// TIA Portal project "Stack_v000_000_005" (V16)
// 000_000_001: create project
// 000_000_002: create Stack.Add
// 000_000_003: create Stack.Remove
// 000_000_004: create Stack.Clear
// 000_000_005: create Stack
// 000_000_006: validation
// 001_000_000: release

(* hardware
DEVICE "S7-1200 station_1"  S7-1200 Station
   slot 0: "Rack_0"  S7-1200 Rack  Rack  V1.0
   slot 1: "PLC_1"  CPU 1212C DC/DC/DC  6ES7 212-1AE40-0XB0  V4.4
*)

// ===== PLC "PLC_1"  CPU 1212C DC/DC/DC =====

VAR_GLOBAL   // PLC tag table "Default tag table"
   "System_Byte" AT %MB1 : Byte;
   "FirstScan" AT %M1.0 : Bool;
   "DiagStatusUpdate" AT %M1.1 : Bool;
   "AlwaysTRUE" AT %M1.2 : Bool;
   "AlwaysFALSE" AT %M1.3 : Bool;
   "Clock_Byte" AT %MB0 : Byte;
   "Clock_10Hz" AT %M0.0 : Bool;
   "Clock_5Hz" AT %M0.1 : Bool;
   "Clock_2.5Hz" AT %M0.2 : Bool;
   "Clock_2Hz" AT %M0.3 : Bool;
   "Clock_1.25Hz" AT %M0.4 : Bool;
   "Clock_1Hz" AT %M0.5 : Bool;
   "Clock_0.625Hz" AT %M0.6 : Bool;
   "Clock_0.5Hz" AT %M0.7 : Bool;
END_VAR

TYPE "Int[+].UDT"
   STRUCT
      add : DInt;
      data : Array[0..4] of Int;
      length : DInt;
      remove : DInt := -1;
   END_STRUCT;
END_TYPE

TYPE "Stack.Calls.UDT"
   STRUCT
      idle : DInt;
      add : DInt := 1;
      remove : DInt := 2;
      clear : DInt := 3;
   END_STRUCT;
END_TYPE

ORGANIZATION_BLOCK "Main"   // OB1, LAD, ProgramCycle
TITLE = "Main Program Sweep (Cycle)"
{ S7_Optimized_Access := 'TRUE' }
VERSION : 0.1
   VAR_INPUT
      Initial_Call : Bool;   // Initial call of this OB
      Remanence : Bool;   // =True, if remanent data are available
   END_VAR
BEGIN
END_ORGANIZATION_BLOCK

// folder: Stack

FUNCTION_BLOCK "Stack"   // FB1, SCL
TITLE = Stack
{ S7_Optimized_Access := 'TRUE' }
AUTHOR : Machado
FAMILY : Stack
VERSION : 0.1
// calls:
//   idle = 0
//   add = 1
//   remove = 2
//   clear = 3
   VAR_INPUT
      call : DInt;
   END_VAR
   VAR_OUTPUT
      status : String;
   END_VAR
   VAR_IN_OUT
      value : Int;
   END_VAR
   VAR
      buffer : "Int[+].UDT";
      calls : "Stack.Calls.UDT";
   END_VAR
   VAR_TEMP
      message : String;
   END_VAR
   VAR CONSTANT
      IDLE_STATUS_MESSAGE : String := 'idle. no operation.';
      IDLE : DInt;
      ADD : DInt := 1;
      REMOVE : DInt := 2;
      CLEAR : DInt := 3;
      NULL_TOKEN : Int := -100;
      DEFAULT_ADD_INDEX : DInt := 0;
      DEFUALT_REMOVE_INDEX : DInt := -1;
   END_VAR
BEGIN
   CASE #call OF
       #IDLE:
           #message := #IDLE_STATUS_MESSAGE;
       #ADD:
           #message := "Stack.Add"(value := #value,
                                   buffer := #buffer);
       #REMOVE:
           #message := "Stack.Remove"(null_token := #NULL_TOKEN,
                                      value => #value,
                                      buffer := #buffer);
       #CLEAR:
           #message := "Stack.Clear"(default_add_index := #DEFAULT_ADD_INDEX,
                                     default_remove_index := #DEFUALT_REMOVE_INDEX,
                                     null_token := #NULL_TOKEN, buffer := #buffer);
       ELSE
           #message := #IDLE_STATUS_MESSAGE;
   END_CASE;
   #status := #message;
   RETURN;
END_FUNCTION_BLOCK

FUNCTION "Stack.Add" : String   // FC6, SCL
TITLE = Add a Value to the Stack
{ S7_Optimized_Access := 'TRUE' }
AUTHOR : Machado
FAMILY : Stack
VERSION : 0.1
// use [+].Push
// don't use [+].Add
   VAR_INPUT
      value : Int;
   END_VAR
   VAR_IN_OUT
      buffer : "Int[+].UDT";
   END_VAR
BEGIN
   #"Stack.Add" := "Int[+].Push"(value := #value,
                                 buffer := #buffer);
   RETURN;
END_FUNCTION

FUNCTION "Stack.Remove" : String   // FC8, SCL
TITLE = Remove a Value from a Stack
{ S7_Optimized_Access := 'TRUE' }
AUTHOR : Machado
FAMILY : Stack
VERSION : 0.1
// returns value and status message.
// use [+].Pop
// don't us [+].Remove
   VAR_INPUT
      null_token : Int;
   END_VAR
   VAR_OUTPUT
      value : Int;
   END_VAR
   VAR_IN_OUT
      buffer : "Int[+].UDT";
   END_VAR
BEGIN
   #"Stack.Remove" := "Int[+].Pop"(null_token := #null_token,
                                   value => #value,
                                   buffer := #buffer);
   RETURN;
END_FUNCTION

FUNCTION "Stack.Clear" : String   // FC10, SCL
TITLE = Clear All Values from a Stack
{ S7_Optimized_Access := 'TRUE' }
AUTHOR : Machado
FAMILY : Stack
VERSION : 0.1
// returns a string
   VAR_INPUT
      default_add_index : DInt;
      default_remove_index : DInt;
      null_token : Int;
   END_VAR
   VAR_IN_OUT
      buffer : "Int[+].UDT";
   END_VAR
BEGIN
   #"Stack.Clear" := "Int[+].Clear"(default_add_index := #default_add_index,
                                    default_remove_index := #default_remove_index,
                                    null_token := #null_token,
                                    buffer := #buffer);
   RETURN;
END_FUNCTION

// folder: Stack/Int[+]

FUNCTION "Int[+].IsFull" : Bool   // FC1, SCL
TITLE = Array Is Full
{ S7_Optimized_Access := 'TRUE' }
AUTHOR : Machado
FAMILY : Int[+]
VERSION : 0.1
// returns true if array is full
   VAR_INPUT
      buffer : "Int[+].UDT";
   END_VAR
   VAR_TEMP
      size : DInt;
   END_VAR
BEGIN
   #size := UDINT_TO_DINT("Int[].CountOfElements"(#buffer.data));
   IF #buffer.length = #size THEN
       #"Int[+].IsFull" := TRUE;
       RETURN;
   END_IF;
   #"Int[+].IsFull" := FALSE;
   RETURN;
END_FUNCTION

FUNCTION "Int[+].IsEmpty" : Bool   // FC3, SCL
TITLE = Int[+] Data Array Is Empty
{ S7_Optimized_Access := 'TRUE' }
AUTHOR : Machado
FAMILY : Int[+]
VERSION : 0.1
// returns true if array is empty
   VAR_INPUT
      buffer : "Int[+].UDT";
   END_VAR
BEGIN
   IF #buffer.length = 0 THEN
       #"Int[+].IsEmpty" := TRUE;
       RETURN;
   END_IF;
   #"Int[+].IsEmpty" := FALSE;
   RETURN;
END_FUNCTION

FUNCTION "Int[+].Push" : String   // FC4, SCL
TITLE = Push Value Into Data Array
{ S7_Optimized_Access := 'TRUE' }
AUTHOR : Machado
FAMILY : Int[+]
VERSION : 0.1
// dont use push with remove
   VAR_INPUT
      value : Int;
   END_VAR
   VAR_IN_OUT
      buffer : "Int[+].UDT";
   END_VAR
   VAR CONSTANT
      ARRAY_FULL : String := 'array full. no operation.';
      PUSHED : String := 'pushed.';
   END_VAR
BEGIN
   REGION "ARRAY FULL"
       IF "Int[+].IsFull"(#buffer) THEN
           #"Int[+].Push" := #ARRAY_FULL;
           RETURN;
       END_IF;
   END_REGION


   REGION "PUSH"
       #buffer.data[#buffer.add] := #value;
       #buffer.add += 1;
       #buffer.remove += 1;
       #buffer.length += 1;
       #"Int[+].Push" := #PUSHED;
       RETURN;
   END_REGION
END_FUNCTION

FUNCTION "Int[+].Pop" : String   // FC5, SCL
TITLE = Pop a Last Value from Data Array
{ S7_Optimized_Access := 'TRUE' }
AUTHOR : Machado
FAMILY : Int[+]
VERSION : 0.1
// do not use with Add
   VAR_INPUT
      null_token : Int;
   END_VAR
   VAR_OUTPUT
      value : Int;
   END_VAR
   VAR_IN_OUT
      buffer : "Int[+].UDT";
   END_VAR
   VAR CONSTANT
      ARRAY_EMPTY : String := 'array empty. no operation.';
      POPPED : String := 'popped';
   END_VAR
BEGIN
   REGION "ARRAY EMPTY"
       IF "Int[+].IsEmpty"(#buffer) THEN
           #value := #null_token;
           #"Int[+].Pop" := #ARRAY_EMPTY;
           RETURN;
       END_IF;
   END_REGION


   REGION "POP"
       #value := #buffer.data[#buffer.remove];
       #buffer.data[#buffer.remove] := #null_token;
       #buffer.add -= 1;
       #buffer.remove -= 1;
       #buffer.length -= 1;
       #"Int[+].Pop" := #POPPED;
       RETURN;
   END_REGION
END_FUNCTION

FUNCTION "Int[+].Clear" : String   // FC9, SCL
{ S7_Optimized_Access := 'TRUE' }
AUTHOR : Machado
FAMILY : Int[+]
VERSION : 0.1
   VAR_INPUT
      default_add_index : DInt;
      default_remove_index : DInt;
      null_token : Int;
   END_VAR
   VAR_IN_OUT
      buffer : "Int[+].UDT";
   END_VAR
   VAR_TEMP
      i : DInt;
      size : DInt;
   END_VAR
   VAR CONSTANT
      DONE : String := 'cleared.';
   END_VAR
BEGIN
   REGION "GET SIZE"
       #size := UDINT_TO_DINT("Int[].CountOfElements"(#buffer.data));
   END_REGION

   REGION "CLEAR DATA"
       FOR #i := 0 TO #size - 1 DO
           #buffer.data[#i] := #null_token;
       END_FOR;
   END_REGION

   REGION "CLEAR META DATA"
       #buffer.add := #default_add_index;
       #buffer.remove := #default_remove_index;
       #buffer.length := 0;
   END_REGION

   REGION "RETURN"
       #"Int[+].Clear" := #DONE;
       RETURN;
   END_REGION
END_FUNCTION

// folder: Stack/Int[+]/DInt

FUNCTION "DInt.RolloverIncrement" : DInt   // FC7, SCL
TITLE = Increments a Value with Rollover
{ S7_Optimized_Access := 'TRUE' }
AUTHOR : Machado
FAMILY : DInt
VERSION : 0.1
   VAR_INPUT
      value : DInt;
      rollover : DInt;
   END_VAR
BEGIN
   #"DInt.RolloverIncrement" := (#value + 1) MOD #rollover;
   RETURN;
END_FUNCTION

// folder: Stack/Int[+]/Int[]

FUNCTION "Int[].CountOfElements" : UDInt   // FC2, SCL
{ S7_Optimized_Access := 'TRUE' }
VERSION : 0.1
   VAR_INPUT
      data : Variant;
   END_VAR
BEGIN
   #"Int[].CountOfElements" := CountOfElements(#data);
   RETURN;
END_FUNCTION